(* PLC project Motor start stop latch, react-plc-diagram PLCopen XML test fixtures 0.1.0 *)
(* stored: creationDateTime 2026-08-12T00:00:00Z, modificationDateTime 2026-08-12T00:00:00Z *)

PROGRAM MotorLatch
  VAR
    Stop : BOOL;
    Start : BOOL;
    Motor : BOOL;
  END_VAR

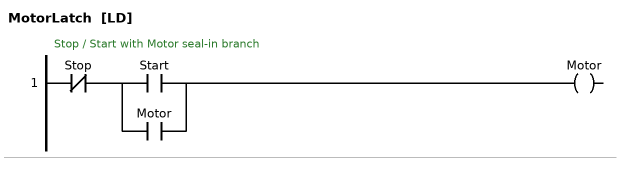
(* LD diagram, written out as Structured Text *)
(* Stop / Start with Motor seal-in branch *)
Motor := NOT Stop AND (Start OR Motor);
END_PROGRAM
